{attribute 'qualified_only'}
VAR_GLOBAL INTERNAL
	{attribute 'ExpandFully'} 
	// Fixed-size array to store all signal-receiver entries.
	// Index 0 is reserved and not used (signals with id = 0 are unassigned).
	stEntry				: ARRAY[0..Param.nChannelSize] OF ST_Entry;
	
	// Total number of assigned entries in the stEntry array.
	nAssigned			: UDINT;
END_VAR

(* stored: Version 1.1.0.1
   GVL _Channel: Id {22f7a211-245d-48ea-b392-287640146104} *)
